Universal Robots PolyScope program: grpB.urp

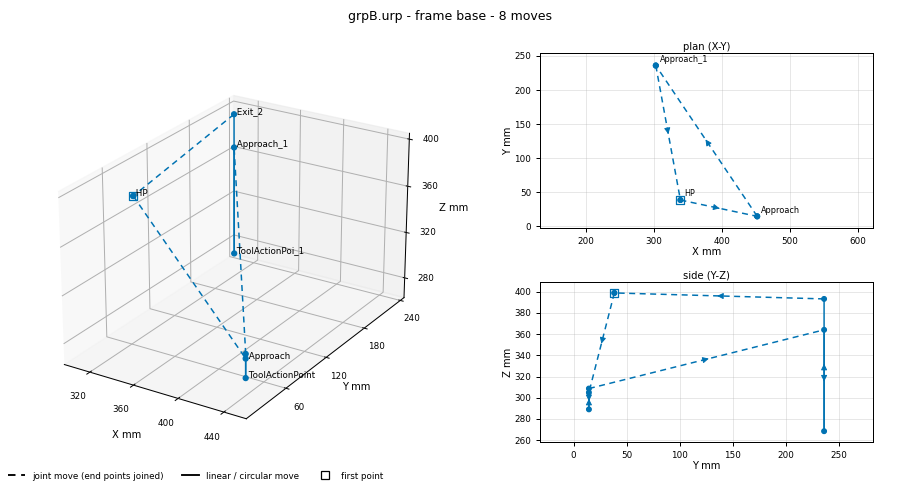
[picture p0: tool path of grpB.urp in frame base, 8 of 8 moves have a stored position in this frame; points joined in program order, loops and branches not executed]
Program grpB (installation=default directory=/programs/Students createdIn=5.11.9.1010452 lastSavedIn=5.11.9.1010452 robotSerialNumber=20225200364)
Calibrated DH parameters: a=[0.00002, -0.569483, -0.54992, -0.00001, -0.000036, 0]; d=[0.180894, -146.691669, 192.918669, -46.053088, 0.119778, 0.115602]; alpha=[1.571425, -0.001534, 0.003359, 1.568739, -1.571477, 0]; deltaTheta=[0, 0.376258, -0.101074, -0.275185, -0.000002, 0]
Robot Program (runOnlyOnce=false)
  URCap RG Grip (OnRobot, OnRobot A/S) dataModel(rg-target-force=40.0, rg-target-width=0.1, Variable(key=on_return, variable(name=on_return)))
  MoveJ speed 60 deg/s, acceleration 80 deg/s^2 (useActiveTCP=true) feature=Base
    Waypoint HP: TCP in base x=339.401 y=38.316 z=398.781 mm, rx=2.2309 ry=-2.1852 rz=-0.032 rad; joints [36.729, -82.18, -126.752, -242.339, -91.192, -144.236] deg
    Loop Counting (count=6) loopVariable(name=Loop_1)
      URCap Palletizing (polyscope-pallet-impl, Universal Robots) dataModel(palletFeature=Base, isPalletizing=false, Variable(key=name, variable(name=Pallet_1)), Variable(key=globalCountingVariable, variable(name=Pallet_1_cnt_1, initializeExpression=1)), Variable(key=layerNumberVariable, variable(name=Pallet_1_lno, initializeExpression=1)), Variable(key=layerCountingVariable, variable(name=Pallet_1_lct, initializeExpression=1)), Variable(key=handleSeparatorVariable, variable(name=Pallet_1_sep, initializeExpression=False)), Variable(key=totalCountVariable, variable(name=Pallet_1_tct, initializeExpression=1)), Variable(key=referencePoint, variable(featureName=referencePoint)), Variable(key=separatorPoint, variable(featureName=separatorPoint)), Length(key=objectHeight value=0.015 unit=M)); state(isChildrenLocked=true)
        URCap Patterns (polyscope-pallet-impl, Universal Robots) state(isChildrenLocked=true)
          URCap Pattern (polyscope-pallet-impl, Universal Robots) dataModel(UUID=368b9eff-c81a-4cc4-85a8-2659ca26b315, patternType=LINE, objects=2, Variable(key=nameVariable, variable(name=Line_Pattern_1))); state(isChildrenLocked=true)
            URCap Item (polyscope-pallet-impl, Universal Robots) dataModel(UUID=9a3704ec-8d27-4c4b-a56d-25a0d66e6629, patternType=LINE, index=0, calibrationDeltaTheta=[-2.1094217540068572E-7, 0.37625772532806073, -0.10107441100396769, -0.2751850025766889, -1.8024952768980196E-6, 2.9402326063437956E-8], calibrationA=[2.0416891277915125E-5, -0.5694828868469309, -0.5499202125525207, -9.504674691390763E-6, -3.603723657207661E-5, 0.0], calibrationD=[0.1808937726775539, -146.69166934821124, 192.91866861971778, -46.05308757405963, 0.11977780403821288, 0.11560212559305974], calibrationAlpha=[1.5714252480212174, -0.0015337665762078037, 0.0033588312559612306, 1.5687392298942362, -1.5714772428732047, 0.0], calibrationJointChecksum=[-1490546360, -1456574554, -1506622700, -1493399207, -1492840923, -1492940558], calibrationStatus=2, calibrationValidChecksum=true, baseToFeature=[0.0, 0.0, 0.0, 0.0, 0.0, 0.0], TCPOffset=[2.6868845456327114E-6, 3.218907108143432E-5, 1.988572699768154E-5, -1.138352401362983E-4, 2.3773279093772227E-5, 3.3708227174379763E-6], Variable(key=variable, variable(name=StartItem_1)), JointPositions(key=jointpositions, JointPosition(key=[1], Angle(key=pos value=0.419802 unit=RAD)), JointPosition(key=[2], Angle(key=pos value=-1.809951 unit=RAD)), JointPosition(key=[3], Angle(key=pos value=-2.12005 unit=RAD)), JointPosition(key=[4], Angle(key=pos value=-3.960683 unit=RAD)), JointPosition(key=[5], Angle(key=pos value=-1.586707 unit=RAD)), JointPosition(key=[6], Angle(key=pos value=-2.746237 unit=RAD))))
            URCap Item (polyscope-pallet-impl, Universal Robots) dataModel(UUID=52f99ad6-588a-4c4c-82d0-046d1d96f193, patternType=LINE, index=1, calibrationDeltaTheta=[-2.1094217540068572E-7, 0.37625772532806073, -0.10107441100396769, -0.2751850025766889, -1.8024952768980196E-6, 2.9402326063437956E-8], calibrationA=[2.0416891277915125E-5, -0.5694828868469309, -0.5499202125525207, -9.504674691390763E-6, -3.603723657207661E-5, 0.0], calibrationD=[0.1808937726775539, -146.69166934821124, 192.91866861971778, -46.05308757405963, 0.11977780403821288, 0.11560212559305974], calibrationAlpha=[1.5714252480212174, -0.0015337665762078037, 0.0033588312559612306, 1.5687392298942362, -1.5714772428732047, 0.0], calibrationJointChecksum=[-1490546360, -1456574554, -1506622700, -1493399207, -1492840923, -1492940558], calibrationStatus=2, calibrationValidChecksum=true, baseToFeature=[0.0, 0.0, 0.0, 0.0, 0.0, 0.0], TCPOffset=[-1.1233085088669216E-5, 1.773362738044515E-6, 4.0124967435328784E-6, -7.304529472293159E-6, -6.067439158460444E-6, 2.488920498882956E-6], Variable(key=variable, variable(name=EndItem_1)), JointPositions(key=jointpositions, JointPosition(key=[1], Angle(key=pos value=0.398383 unit=RAD)), JointPosition(key=[2], Angle(key=pos value=-1.844105 unit=RAD)), JointPosition(key=[3], Angle(key=pos value=-2.072895 unit=RAD)), JointPosition(key=[4], Angle(key=pos value=-3.973966 unit=RAD)), JointPosition(key=[5], Angle(key=pos value=-1.5859 unit=RAD)), JointPosition(key=[6], Angle(key=pos value=-2.767675 unit=RAD))))
        URCap Layers (polyscope-pallet-impl, Universal Robots) dataModel(separators=[false, false, false], selectedPatterns=[368b9eff-c81a-4cc4-85a8-2659ca26b315, 368b9eff-c81a-4cc4-85a8-2659ca26b315, 368b9eff-c81a-4cc4-85a8-2659ca26b315])
        URCap At Each Item (polyscope-pallet-impl, Universal Robots) dataModel(selectedPattern=368b9eff-c81a-4cc4-85a8-2659ca26b315, selectedPosition=9a3704ec-8d27-4c4b-a56d-25a0d66e6629, Approach_calibrationDeltaTheta=[-2.1094217540068572E-7, 0.37625772532806073, -0.10107441100396769, -0.2751850025766889, -1.8024952768980196E-6, 2.9402326063437956E-8], Approach_calibrationA=[2.0416891277915125E-5, -0.5694828868469309, -0.5499202125525207, -9.504674691390763E-6, -3.603723657207661E-5, 0.0], Approach_calibrationD=[0.1808937726775539, -146.69166934821124, 192.91866861971778, -46.05308757405963, 0.11977780403821288, 0.11560212559305974], Approach_calibrationAlpha=[1.5714252480212174, -0.0015337665762078037, 0.0033588312559612306, 1.5687392298942362, -1.5714772428732047, 0.0], Approach_calibrationJointChecksum=[-1490546360, -1456574554, -1506622700, -1493399207, -1492840923, -1492940558], Approach_calibrationStatus=2, Approach_calibrationValidChecksum=true, Approach_baseToFeature=[0.0, 0.0, 0.0, 0.0, 0.0, 0.0], Approach_TCPOffset=[1.761467848184384E-5, 2.7781053029807268E-5, 1.6800067060063206E-5, -8.989547277361643E-5, -1.7381909268676295E-5, 3.332126419325864E-5], Exit_calibrationDeltaTheta=[-2.1094217540068572E-7, 0.37625772532806073, -0.10107441100396769, -0.2751850025766889, -1.8024952768980196E-6, 2.9402326063437956E-8], Exit_calibrationA=[2.0416891277915125E-5, -0.5694828868469309, -0.5499202125525207, -9.504674691390763E-6, -3.603723657207661E-5, 0.0], Exit_calibrationD=[0.1808937726775539, -146.69166934821124, 192.91866861971778, -46.05308757405963, 0.11977780403821288, 0.11560212559305974], Exit_calibrationAlpha=[1.5714252480212174, -0.0015337665762078037, 0.0033588312559612306, 1.5687392298942362, -1.5714772428732047, 0.0], Exit_calibrationJointChecksum=[-1490546360, -1456574554, -1506622700, -1493399207, -1492840923, -1492940558], Exit_calibrationStatus=2, Exit_calibrationValidChecksum=true, Exit_baseToFeature=[0.0, 0.0, 0.0, 0.0, 0.0, 0.0], Exit_TCPOffset=[3.582266093114252E-6, -1.155257506713081E-6, 3.988152352973895E-6, -3.160951924481522E-5, -1.5140422987903268E-5, -2.403678189092286E-5], currentWizardState=LANDING, Pose(key=refBaseToFeature, Position(key=posePosition, Length(key=X value=0 unit=M), Length(key=Y value=0 unit=M), Length(key=Z value=0 unit=M)), Rotation(key=poseRotation, Angle(key=RX value=0 unit=RAD), Angle(key=RY value=0 unit=RAD), Angle(key=RZ value=0 unit=RAD))), Pose(key=refPose, Position(key=posePosition, Length(key=X value=0.452251 unit=M), Length(key=Y value=0.014358 unit=M), Length(key=Z value=0.289056 unit=M)), Rotation(key=poseRotation, Angle(key=RX value=2.238278 unit=RAD), Angle(key=RY value=-2.171608 unit=RAD), Angle(key=RZ value=-0.027778 unit=RAD))), JointPositions(key=Approach_jointpositions, JointPosition(key=[1], Angle(key=pos value=0.42473 unit=RAD)), JointPosition(key=[2], Angle(key=pos value=-1.740044 unit=RAD)), JointPosition(key=[3], Angle(key=pos value=-2.100953 unit=RAD)), JointPosition(key=[4], Angle(key=pos value=-4.041414 unit=RAD)), JointPosition(key=[5], Angle(key=pos value=-1.581802 unit=RAD)), JointPosition(key=[6], Angle(key=pos value=-2.742355 unit=RAD))), JointPositions(key=Exit_jointpositions, JointPosition(key=[1], Angle(key=pos value=0.424724 unit=RAD)), JointPosition(key=[2], Angle(key=pos value=-1.735522 unit=RAD)), JointPosition(key=[3], Angle(key=pos value=-2.098004 unit=RAD)), JointPosition(key=[4], Angle(key=pos value=-4.048884 unit=RAD)), JointPosition(key=[5], Angle(key=pos value=-1.581818 unit=RAD)), JointPosition(key=[6], Angle(key=pos value=-2.742386 unit=RAD))))
          URCap Generated Movements (polyscope-pallet-impl, Universal Robots) state(isChildrenLocked=true)
            MoveJ speed 60 deg/s, acceleration 80 deg/s^2 (useActiveTCP=true) feature=referencePoint
              Waypoint Approach: TCP in base x=452.223 y=14.34 z=304.926 mm, rx=2.2382 ry=-2.1716 rz=-0.0279 rad; joints [24.334, -99.697, -120.379, -231.557, -90.633, -157.125] deg; TCP offset x=0 y=0 z=0 mm, rx=0 ry=0 rz=0 rad; feature pose in base x=452.251 y=14.358 z=289.056 mm, rx=2.2383 ry=-2.1716 rz=-0.0278 rad
            MoveL speed 250 mm/s, acceleration 1200 mm/s^2 (useActiveTCP=true) feature(featureName=referencePoint)
              Waypoint ToolActionPoint: TCP in base x=452.251 y=14.358 z=289.056 mm, rx=2.2383 ry=-2.1716 rz=-0.0278 rad; joints [24.337, -100.828, -121.067, -229.734, -90.626, -157.118] deg; TCP offset x=0 y=0 z=0 mm, rx=0 ry=0 rz=0 rad
            Folder Tool action
              URCap RG Grip (OnRobot, OnRobot A/S) dataModel(rg-target-force=40.0, rg-target-width=0.07540000000000001)
            MoveL speed 250 mm/s, acceleration 1200 mm/s^2 (useActiveTCP=true) feature(featureName=referencePoint)
              Waypoint Exit_1: TCP in base x=452.252 y=14.355 z=308.678 mm, rx=2.2383 ry=-2.1716 rz=-0.0278 rad; joints [24.334, -99.439, -120.207, -231.985, -90.633, -157.129] deg; TCP offset x=0 y=0 z=0 mm, rx=0 ry=0 rz=0 rad
      URCap Palletizing (polyscope-pallet-impl, Universal Robots) dataModel(palletFeature=Base, isPalletizing=true, Variable(key=name, variable(name=Pallet_2)), Variable(key=globalCountingVariable, variable(name=Pallet_2_cnt, initializeExpression=1)), Variable(key=layerNumberVariable, variable(name=Pallet_2_lno, initializeExpression=1)), Variable(key=layerCountingVariable, variable(name=Pallet_2_lct, initializeExpression=1)), Variable(key=handleSeparatorVariable, variable(name=Pallet_2_sep, initializeExpression=False)), Variable(key=totalCountVariable, variable(name=Pallet_2_tct, initializeExpression=1)), Variable(key=referencePoint, variable(featureName=referencePoin_1)), Variable(key=separatorPoint, variable(featureName=separatorPoin_1)), Length(key=objectHeight value=0.015 unit=M)); state(isChildrenLocked=true)
        URCap Patterns (polyscope-pallet-impl, Universal Robots) state(isChildrenLocked=true)
          URCap Pattern (polyscope-pallet-impl, Universal Robots) dataModel(UUID=d9a7a4ad-0665-4455-a2d0-a41ab3c0d793, patternType=LINE, objects=2, Variable(key=nameVariable, variable(name=Line_Pattern_2))); state(isChildrenLocked=true)
            URCap Item (polyscope-pallet-impl, Universal Robots) dataModel(UUID=0a3d0043-4615-43b5-9a77-a8b26f42fe14, patternType=LINE, index=0, calibrationDeltaTheta=[-2.1094217540068572E-7, 0.37625772532806073, -0.10107441100396769, -0.2751850025766889, -1.8024952768980196E-6, 2.9402326063437956E-8], calibrationA=[2.0416891277915125E-5, -0.5694828868469309, -0.5499202125525207, -9.504674691390763E-6, -3.603723657207661E-5, 0.0], calibrationD=[0.1808937726775539, -146.69166934821124, 192.91866861971778, -46.05308757405963, 0.11977780403821288, 0.11560212559305974], calibrationAlpha=[1.5714252480212174, -0.0015337665762078037, 0.0033588312559612306, 1.5687392298942362, -1.5714772428732047, 0.0], calibrationJointChecksum=[-1490546360, -1456574554, -1506622700, -1493399207, -1492840923, -1492940558], calibrationStatus=2, calibrationValidChecksum=true, baseToFeature=[0.0, 0.0, 0.0, 0.0, 0.0, 0.0], TCPOffset=[1.2018683137271502E-5, 1.2898918078319E-5, 3.2929703053019566E-5, -1.4272770987504921E-5, 1.2116891347895457E-5, -1.797819080023642E-5], Variable(key=variable, variable(name=StartItem_2)), JointPositions(key=jointpositions, JointPosition(key=[1], Angle(key=pos value=1.124181 unit=RAD)), JointPosition(key=[2], Angle(key=pos value=-1.677054 unit=RAD)), JointPosition(key=[3], Angle(key=pos value=-2.260117 unit=RAD)), JointPosition(key=[4], Angle(key=pos value=-3.933363 unit=RAD)), JointPosition(key=[5], Angle(key=pos value=-1.597693 unit=RAD)), JointPosition(key=[6], Angle(key=pos value=-2.042694 unit=RAD))))
            URCap Item (polyscope-pallet-impl, Universal Robots) dataModel(UUID=2278e55f-7ae9-4ebe-9340-457ba648b36e, patternType=LINE, index=1, calibrationDeltaTheta=[-2.1094217540068572E-7, 0.37625772532806073, -0.10107441100396769, -0.2751850025766889, -1.8024952768980196E-6, 2.9402326063437956E-8], calibrationA=[2.0416891277915125E-5, -0.5694828868469309, -0.5499202125525207, -9.504674691390763E-6, -3.603723657207661E-5, 0.0], calibrationD=[0.1808937726775539, -146.69166934821124, 192.91866861971778, -46.05308757405963, 0.11977780403821288, 0.11560212559305974], calibrationAlpha=[1.5714252480212174, -0.0015337665762078037, 0.0033588312559612306, 1.5687392298942362, -1.5714772428732047, 0.0], calibrationJointChecksum=[-1490546360, -1456574554, -1506622700, -1493399207, -1492840923, -1492940558], calibrationStatus=2, calibrationValidChecksum=true, baseToFeature=[0.0, 0.0, 0.0, 0.0, 0.0, 0.0], TCPOffset=[3.16417898940935E-5, 2.6172659556844557E-6, -7.331736447235837E-6, 1.333391651039793E-5, -1.1496433426125451E-5, 6.149251622774298E-5], Variable(key=variable, variable(name=EndItem_2)), JointPositions(key=jointpositions, JointPosition(key=[1], Angle(key=pos value=1.207982 unit=RAD)), JointPosition(key=[2], Angle(key=pos value=-1.636595 unit=RAD)), JointPosition(key=[3], Angle(key=pos value=-2.305171 unit=RAD)), JointPosition(key=[4], Angle(key=pos value=-3.926681 unit=RAD)), JointPosition(key=[5], Angle(key=pos value=-1.598967 unit=RAD)), JointPosition(key=[6], Angle(key=pos value=-1.958923 unit=RAD))))
        URCap Layers (polyscope-pallet-impl, Universal Robots) dataModel(separators=[false, false, false], selectedPatterns=[d9a7a4ad-0665-4455-a2d0-a41ab3c0d793, d9a7a4ad-0665-4455-a2d0-a41ab3c0d793, d9a7a4ad-0665-4455-a2d0-a41ab3c0d793])
        URCap At Each Item (polyscope-pallet-impl, Universal Robots) dataModel(selectedPattern=d9a7a4ad-0665-4455-a2d0-a41ab3c0d793, selectedPosition=0a3d0043-4615-43b5-9a77-a8b26f42fe14, Approach_calibrationDeltaTheta=[-2.1094217540068572E-7, 0.37625772532806073, -0.10107441100396769, -0.2751850025766889, -1.8024952768980196E-6, 2.9402326063437956E-8], Approach_calibrationA=[2.0416891277915125E-5, -0.5694828868469309, -0.5499202125525207, -9.504674691390763E-6, -3.603723657207661E-5, 0.0], Approach_calibrationD=[0.1808937726775539, -146.69166934821124, 192.91866861971778, -46.05308757405963, 0.11977780403821288, 0.11560212559305974], Approach_calibrationAlpha=[1.5714252480212174, -0.0015337665762078037, 0.0033588312559612306, 1.5687392298942362, -1.5714772428732047, 0.0], Approach_calibrationJointChecksum=[-1490546360, -1456574554, -1506622700, -1493399207, -1492840923, -1492940558], Approach_calibrationStatus=2, Approach_calibrationValidChecksum=true, Approach_baseToFeature=[0.0, 0.0, 0.0, 0.0, 0.0, 0.0], Approach_TCPOffset=[-1.0252083862682948E-5, -1.0985974046584523E-6, 4.721684620845323E-6, -1.601007812302085E-5, 4.2221409929860464E-5, -2.0644725078100677E-5], Exit_calibrationDeltaTheta=[-2.1094217540068572E-7, 0.37625772532806073, -0.10107441100396769, -0.2751850025766889, -1.8024952768980196E-6, 2.9402326063437956E-8], Exit_calibrationA=[2.0416891277915125E-5, -0.5694828868469309, -0.5499202125525207, -9.504674691390763E-6, -3.603723657207661E-5, 0.0], Exit_calibrationD=[0.1808937726775539, -146.69166934821124, 192.91866861971778, -46.05308757405963, 0.11977780403821288, 0.11560212559305974], Exit_calibrationAlpha=[1.5714252480212174, -0.0015337665762078037, 0.0033588312559612306, 1.5687392298942362, -1.5714772428732047, 0.0], Exit_calibrationJointChecksum=[-1490546360, -1456574554, -1506622700, -1493399207, -1492840923, -1492940558], Exit_calibrationStatus=2, Exit_calibrationValidChecksum=true, Exit_baseToFeature=[0.0, 0.0, 0.0, 0.0, 0.0, 0.0], Exit_TCPOffset=[3.031500758254868E-6, 8.589234255174105E-6, 6.132106393663683E-6, -4.678619103192354E-5, 4.767019059137122E-5, -1.5113320905268102E-5], currentWizardState=LANDING, Pose(key=refBaseToFeature, Position(key=posePosition, Length(key=X value=0 unit=M), Length(key=Y value=0 unit=M), Length(key=Z value=0 unit=M)), Rotation(key=poseRotation, Angle(key=RX value=0 unit=RAD), Angle(key=RY value=0 unit=RAD), Angle(key=RZ value=0 unit=RAD))), Pose(key=refPose, Position(key=posePosition, Length(key=X value=0.303222 unit=M), Length(key=Y value=0.235983 unit=M), Length(key=Z value=0.268485 unit=M)), Rotation(key=poseRotation, Angle(key=RX value=2.238284 unit=RAD), Angle(key=RY value=-2.171575 unit=RAD), Angle(key=RZ value=-0.027781 unit=RAD))), JointPositions(key=Approach_jointpositions, JointPosition(key=[1], Angle(key=pos value=1.123941 unit=RAD)), JointPosition(key=[2], Angle(key=pos value=-1.552782 unit=RAD)), JointPosition(key=[3], Angle(key=pos value=-2.174946 unit=RAD)), JointPosition(key=[4], Angle(key=pos value=-4.142846 unit=RAD)), JointPosition(key=[5], Angle(key=pos value=-1.598149 unit=RAD)), JointPosition(key=[6], Angle(key=pos value=-2.043665 unit=RAD))), JointPositions(key=Exit_jointpositions, JointPosition(key=[1], Angle(key=pos value=1.123854 unit=RAD)), JointPosition(key=[2], Angle(key=pos value=-1.52272 unit=RAD)), JointPosition(key=[3], Angle(key=pos value=-2.143777 unit=RAD)), JointPosition(key=[4], Angle(key=pos value=-4.204083 unit=RAD)), JointPosition(key=[5], Angle(key=pos value=-1.598243 unit=RAD)), JointPosition(key=[6], Angle(key=pos value=-2.04397 unit=RAD))))
          URCap Generated Movements (polyscope-pallet-impl, Universal Robots) state(isChildrenLocked=true)
            MoveJ speed 60 deg/s, acceleration 80 deg/s^2 (useActiveTCP=true) feature=referencePoin_1
              Waypoint Approach_1: TCP in base x=303.223 y=235.993 z=364.021 mm, rx=2.2383 ry=-2.1715 rz=-0.0278 rad; joints [64.398, -88.97, -124.615, -237.369, -91.567, -117.094] deg; TCP offset x=0 y=0 z=0 mm, rx=0 ry=0 rz=0 rad; feature pose in base x=303.222 y=235.983 z=268.485 mm, rx=2.2383 ry=-2.1716 rz=-0.0278 rad
            MoveL speed 250 mm/s, acceleration 1200 mm/s^2 (useActiveTCP=true) feature(featureName=referencePoin_1)
              Waypoint ToolActionPoi_1: TCP in base x=303.222 y=235.983 z=268.485 mm, rx=2.2383 ry=-2.1716 rz=-0.0278 rad; joints [64.412, -96.09, -129.498, -225.361, -91.541, -117.038] deg; TCP offset x=0 y=0 z=0 mm, rx=0 ry=0 rz=0 rad
            Folder Tool action
              URCap RG Grip (OnRobot, OnRobot A/S) dataModel(rg-target-force=40.0, rg-target-width=0.10070000000000001)
            MoveL speed 250 mm/s, acceleration 1200 mm/s^2 (useActiveTCP=true) feature(featureName=referencePoin_1)
              Waypoint Exit_2: TCP in base x=303.213 y=235.98 z=393.152 mm, rx=2.2383 ry=-2.1715 rz=-0.0278 rad; joints [64.393, -87.246, -122.83, -240.878, -91.574, -117.111] deg; TCP offset x=0 y=0 z=0 mm, rx=0 ry=0 rz=0 rad
    Waypoint HP: TCP in base x=339.401 y=38.316 z=398.781 mm, rx=2.2309 ry=-2.1852 rz=-0.032 rad; joints [36.729, -82.18, -126.752, -242.339, -91.192, -144.236] deg
    Halt
